// TIA Portal V20 export
TYPE "LER_typePartDataEm4"
// stored: Access Published
   STRUCT
      anodeMainPnP1 : "LER_typePartData";
      anodeAlignTable : "LER_typePartData";
      anodeMainPnP2 : "LER_typePartData";
      anodeAlignVision : "LER_typeVisionAlignData";
   END_STRUCT;
END_TYPE
